// Mitsubishi GX Works2 project: 04-06-2020 PWM   PLC: FX3U/FX3UC

PROGRAM MAIN
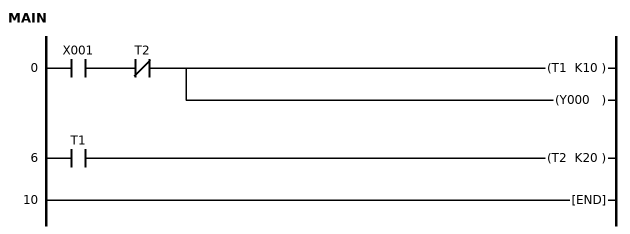
0     LD      X001
      ANI     T2
      OUT     T1 K10
      OUT     Y000
6     LD      T1
      OUT     T2 K20
10    END
END_PROGRAM
